INTERFACE I_StepWorker

METHOD PUBLIC mAddCondition : I_StepWorker
VAR_INPUT
	itfStepCondition : I_StepCondition;
END_VAR
END_METHOD

END_INTERFACE

(* stored: Version 1.1.0.1, ProductVersion 3.1.4024.0
   Itf I_StepWorker: Id {6e16077e-14a2-4353-85e5-4c73ddfcb1e4}
   Method mAddCondition: Id {22238d22-4d9e-4af6-9b13-3aa58c4ea183} *)
